// TIA Portal V16 export
// export: Created 2022-09-01T13:58:51.8751528Z, ExportSetting WithDefaults, DisplayName Totally Integrated Automation Portal, DisplayVersion V16, DisplayName TIA Portal Version Control Interface, DisplayVersion V16, DisplayName TIA Portal Openness, DisplayVersion V16, DisplayName STEP 7 Professional, DisplayVersion V16, DisplayName STEP 7 Safety, DisplayVersion V16, DisplayName WinCC Advanced, DisplayVersion V16
FUNCTION "Saídas_EV_Filt2" : Void   // FC5, LAD
{ S7_Optimized_Access := 'TRUE' }
VERSION : 0.1
// stored: AutoNumber true, IsIECCheckEnabled false, SetENOAutomatically false, UDAEnableTagReadback false
BEGIN

REGION Network 1
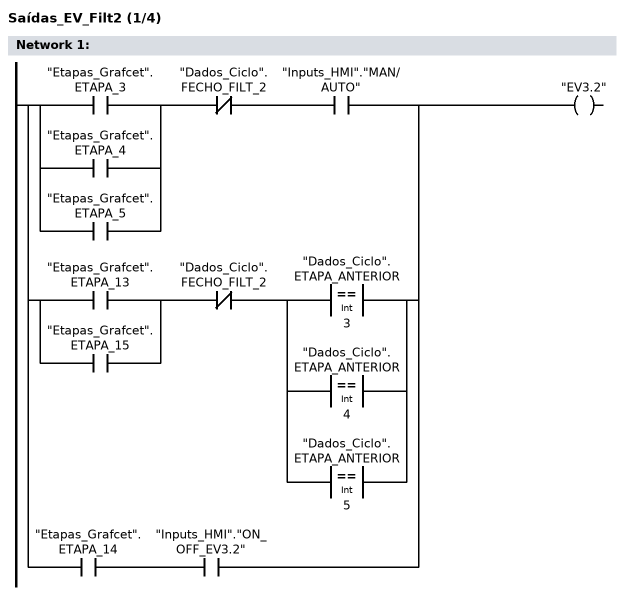
   RUNG wire#powerrail
      Contact( "Etapas_Grafcet".ETAPA_3 )
      wire#w1
      I_Contact( "Dados_Ciclo".FECHO_FILT_2 )
      Contact( "Inputs_HMI"."MAN/AUTO" )
      wire#w2
      Coil( "EV3.2" )
   END_RUNG
   RUNG wire#powerrail
      Contact( "Etapas_Grafcet".ETAPA_4 )
   END_RUNG wire#w1
   RUNG wire#powerrail
      Contact( "Etapas_Grafcet".ETAPA_5 )
   END_RUNG wire#w1
   RUNG wire#powerrail
      Contact( "Etapas_Grafcet".ETAPA_13 )
      wire#w3
      I_Contact( "Dados_Ciclo".FECHO_FILT_2 )
      wire#w4
      { S7_Templates := "SrcType := Int" } EQ_Contact(in1 := "Dados_Ciclo".ETAPA_ANTERIOR, in2 := 3)
   END_RUNG wire#w2
   RUNG wire#powerrail
      Contact( "Etapas_Grafcet".ETAPA_15 )
   END_RUNG wire#w3
   RUNG wire#w4
      { S7_Templates := "SrcType := Int" } EQ_Contact(in1 := "Dados_Ciclo".ETAPA_ANTERIOR, in2 := 4)
   END_RUNG wire#w2
   RUNG wire#w4
      { S7_Templates := "SrcType := Int" } EQ_Contact(in1 := "Dados_Ciclo".ETAPA_ANTERIOR, in2 := 5)
   END_RUNG wire#w2
   RUNG wire#powerrail
      Contact( "Etapas_Grafcet".ETAPA_14 )
      Contact( "Inputs_HMI"."ON_OFF_EV3.2" )
   END_RUNG wire#w2
   // the same network as SCL:
   "EV3.2" := (("Etapas_Grafcet".ETAPA_3 OR "Etapas_Grafcet".ETAPA_4 OR "Etapas_Grafcet".ETAPA_5) AND NOT "Dados_Ciclo".FECHO_FILT_2 AND "Inputs_HMI"."MAN/AUTO") OR (("Etapas_Grafcet".ETAPA_13 OR "Etapas_Grafcet".ETAPA_15) AND NOT "Dados_Ciclo".FECHO_FILT_2 AND (("Dados_Ciclo".ETAPA_ANTERIOR = 3) OR ("Dados_Ciclo".ETAPA_ANTERIOR = 4) OR ("Dados_Ciclo".ETAPA_ANTERIOR = 5))) OR ("Etapas_Grafcet".ETAPA_14 AND "Inputs_HMI"."ON_OFF_EV3.2");
END_REGION

REGION Network 2
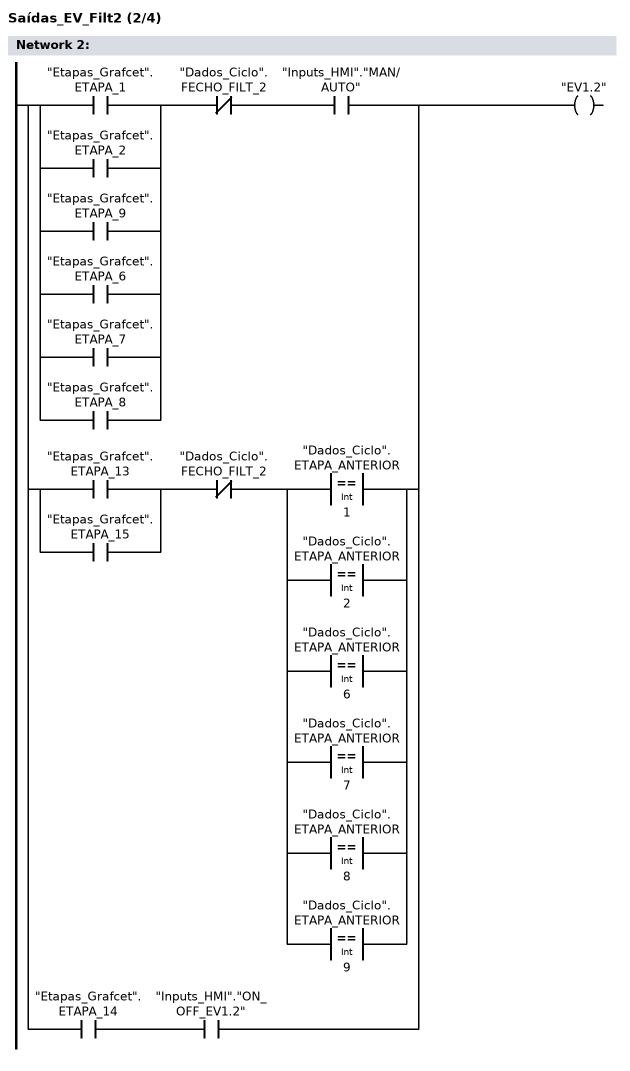
   RUNG wire#powerrail
      Contact( "Etapas_Grafcet".ETAPA_1 )
      wire#w1
      I_Contact( "Dados_Ciclo".FECHO_FILT_2 )
      Contact( "Inputs_HMI"."MAN/AUTO" )
      wire#w2
      Coil( "EV1.2" )
   END_RUNG
   RUNG wire#powerrail
      Contact( "Etapas_Grafcet".ETAPA_2 )
   END_RUNG wire#w1
   RUNG wire#powerrail
      Contact( "Etapas_Grafcet".ETAPA_9 )
   END_RUNG wire#w1
   RUNG wire#powerrail
      Contact( "Etapas_Grafcet".ETAPA_6 )
   END_RUNG wire#w1
   RUNG wire#powerrail
      Contact( "Etapas_Grafcet".ETAPA_7 )
   END_RUNG wire#w1
   RUNG wire#powerrail
      Contact( "Etapas_Grafcet".ETAPA_8 )
   END_RUNG wire#w1
   RUNG wire#powerrail
      Contact( "Etapas_Grafcet".ETAPA_13 )
      wire#w3
      I_Contact( "Dados_Ciclo".FECHO_FILT_2 )
      wire#w4
      { S7_Templates := "SrcType := Int" } EQ_Contact(in1 := "Dados_Ciclo".ETAPA_ANTERIOR, in2 := 1)
   END_RUNG wire#w2
   RUNG wire#powerrail
      Contact( "Etapas_Grafcet".ETAPA_15 )
   END_RUNG wire#w3
   RUNG wire#w4
      { S7_Templates := "SrcType := Int" } EQ_Contact(in1 := "Dados_Ciclo".ETAPA_ANTERIOR, in2 := 2)
   END_RUNG wire#w2
   RUNG wire#w4
      { S7_Templates := "SrcType := Int" } EQ_Contact(in1 := "Dados_Ciclo".ETAPA_ANTERIOR, in2 := 6)
   END_RUNG wire#w2
   RUNG wire#w4
      { S7_Templates := "SrcType := Int" } EQ_Contact(in1 := "Dados_Ciclo".ETAPA_ANTERIOR, in2 := 7)
   END_RUNG wire#w2
   RUNG wire#w4
      { S7_Templates := "SrcType := Int" } EQ_Contact(in1 := "Dados_Ciclo".ETAPA_ANTERIOR, in2 := 8)
   END_RUNG wire#w2
   RUNG wire#w4
      { S7_Templates := "SrcType := Int" } EQ_Contact(in1 := "Dados_Ciclo".ETAPA_ANTERIOR, in2 := 9)
   END_RUNG wire#w2
   RUNG wire#powerrail
      Contact( "Etapas_Grafcet".ETAPA_14 )
      Contact( "Inputs_HMI"."ON_OFF_EV1.2" )
   END_RUNG wire#w2
   // the same network as SCL:
   "EV1.2" := (("Etapas_Grafcet".ETAPA_1 OR "Etapas_Grafcet".ETAPA_2 OR "Etapas_Grafcet".ETAPA_9 OR "Etapas_Grafcet".ETAPA_6 OR "Etapas_Grafcet".ETAPA_7 OR "Etapas_Grafcet".ETAPA_8) AND NOT "Dados_Ciclo".FECHO_FILT_2 AND "Inputs_HMI"."MAN/AUTO") OR (("Etapas_Grafcet".ETAPA_13 OR "Etapas_Grafcet".ETAPA_15) AND NOT "Dados_Ciclo".FECHO_FILT_2 AND (("Dados_Ciclo".ETAPA_ANTERIOR = 1) OR ("Dados_Ciclo".ETAPA_ANTERIOR = 2) OR ("Dados_Ciclo".ETAPA_ANTERIOR = 6) OR ("Dados_Ciclo".ETAPA_ANTERIOR = 7) OR ("Dados_Ciclo".ETAPA_ANTERIOR = 8) OR ("Dados_Ciclo".ETAPA_ANTERIOR = 9))) OR ("Etapas_Grafcet".ETAPA_14 AND "Inputs_HMI"."ON_OFF_EV1.2");
END_REGION

REGION Network 3
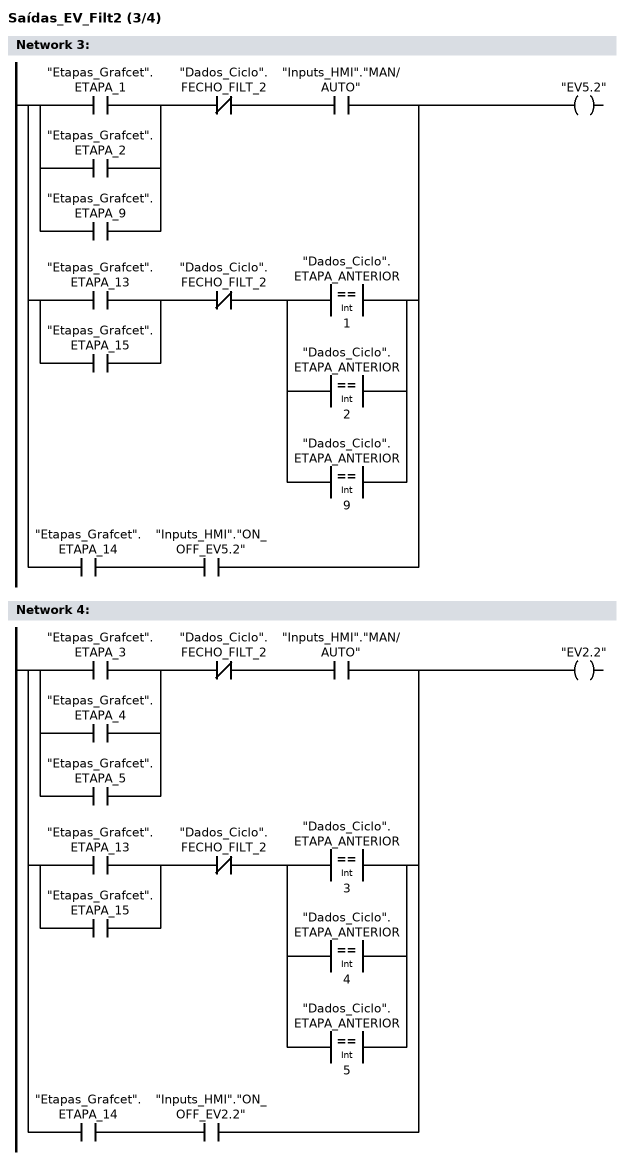
   RUNG wire#powerrail
      Contact( "Etapas_Grafcet".ETAPA_1 )
      wire#w1
      I_Contact( "Dados_Ciclo".FECHO_FILT_2 )
      Contact( "Inputs_HMI"."MAN/AUTO" )
      wire#w2
      Coil( "EV5.2" )
   END_RUNG
   RUNG wire#powerrail
      Contact( "Etapas_Grafcet".ETAPA_2 )
   END_RUNG wire#w1
   RUNG wire#powerrail
      Contact( "Etapas_Grafcet".ETAPA_9 )
   END_RUNG wire#w1
   RUNG wire#powerrail
      Contact( "Etapas_Grafcet".ETAPA_13 )
      wire#w3
      I_Contact( "Dados_Ciclo".FECHO_FILT_2 )
      wire#w4
      { S7_Templates := "SrcType := Int" } EQ_Contact(in1 := "Dados_Ciclo".ETAPA_ANTERIOR, in2 := 1)
   END_RUNG wire#w2
   RUNG wire#powerrail
      Contact( "Etapas_Grafcet".ETAPA_15 )
   END_RUNG wire#w3
   RUNG wire#w4
      { S7_Templates := "SrcType := Int" } EQ_Contact(in1 := "Dados_Ciclo".ETAPA_ANTERIOR, in2 := 2)
   END_RUNG wire#w2
   RUNG wire#w4
      { S7_Templates := "SrcType := Int" } EQ_Contact(in1 := "Dados_Ciclo".ETAPA_ANTERIOR, in2 := 9)
   END_RUNG wire#w2
   RUNG wire#powerrail
      Contact( "Etapas_Grafcet".ETAPA_14 )
      Contact( "Inputs_HMI"."ON_OFF_EV5.2" )
   END_RUNG wire#w2
   // the same network as SCL:
   "EV5.2" := (("Etapas_Grafcet".ETAPA_1 OR "Etapas_Grafcet".ETAPA_2 OR "Etapas_Grafcet".ETAPA_9) AND NOT "Dados_Ciclo".FECHO_FILT_2 AND "Inputs_HMI"."MAN/AUTO") OR (("Etapas_Grafcet".ETAPA_13 OR "Etapas_Grafcet".ETAPA_15) AND NOT "Dados_Ciclo".FECHO_FILT_2 AND (("Dados_Ciclo".ETAPA_ANTERIOR = 1) OR ("Dados_Ciclo".ETAPA_ANTERIOR = 2) OR ("Dados_Ciclo".ETAPA_ANTERIOR = 9))) OR ("Etapas_Grafcet".ETAPA_14 AND "Inputs_HMI"."ON_OFF_EV5.2");
END_REGION

REGION Network 4
   RUNG wire#powerrail
      Contact( "Etapas_Grafcet".ETAPA_3 )
      wire#w1
      I_Contact( "Dados_Ciclo".FECHO_FILT_2 )
      Contact( "Inputs_HMI"."MAN/AUTO" )
      wire#w2
      Coil( "EV2.2" )
   END_RUNG
   RUNG wire#powerrail
      Contact( "Etapas_Grafcet".ETAPA_4 )
   END_RUNG wire#w1
   RUNG wire#powerrail
      Contact( "Etapas_Grafcet".ETAPA_5 )
   END_RUNG wire#w1
   RUNG wire#powerrail
      Contact( "Etapas_Grafcet".ETAPA_13 )
      wire#w3
      I_Contact( "Dados_Ciclo".FECHO_FILT_2 )
      wire#w4
      { S7_Templates := "SrcType := Int" } EQ_Contact(in1 := "Dados_Ciclo".ETAPA_ANTERIOR, in2 := 3)
   END_RUNG wire#w2
   RUNG wire#powerrail
      Contact( "Etapas_Grafcet".ETAPA_15 )
   END_RUNG wire#w3
   RUNG wire#w4
      { S7_Templates := "SrcType := Int" } EQ_Contact(in1 := "Dados_Ciclo".ETAPA_ANTERIOR, in2 := 4)
   END_RUNG wire#w2
   RUNG wire#w4
      { S7_Templates := "SrcType := Int" } EQ_Contact(in1 := "Dados_Ciclo".ETAPA_ANTERIOR, in2 := 5)
   END_RUNG wire#w2
   RUNG wire#powerrail
      Contact( "Etapas_Grafcet".ETAPA_14 )
      Contact( "Inputs_HMI"."ON_OFF_EV2.2" )
   END_RUNG wire#w2
   // the same network as SCL:
   "EV2.2" := (("Etapas_Grafcet".ETAPA_3 OR "Etapas_Grafcet".ETAPA_4 OR "Etapas_Grafcet".ETAPA_5) AND NOT "Dados_Ciclo".FECHO_FILT_2 AND "Inputs_HMI"."MAN/AUTO") OR (("Etapas_Grafcet".ETAPA_13 OR "Etapas_Grafcet".ETAPA_15) AND NOT "Dados_Ciclo".FECHO_FILT_2 AND (("Dados_Ciclo".ETAPA_ANTERIOR = 3) OR ("Dados_Ciclo".ETAPA_ANTERIOR = 4) OR ("Dados_Ciclo".ETAPA_ANTERIOR = 5))) OR ("Etapas_Grafcet".ETAPA_14 AND "Inputs_HMI"."ON_OFF_EV2.2");
END_REGION

REGION Network 5
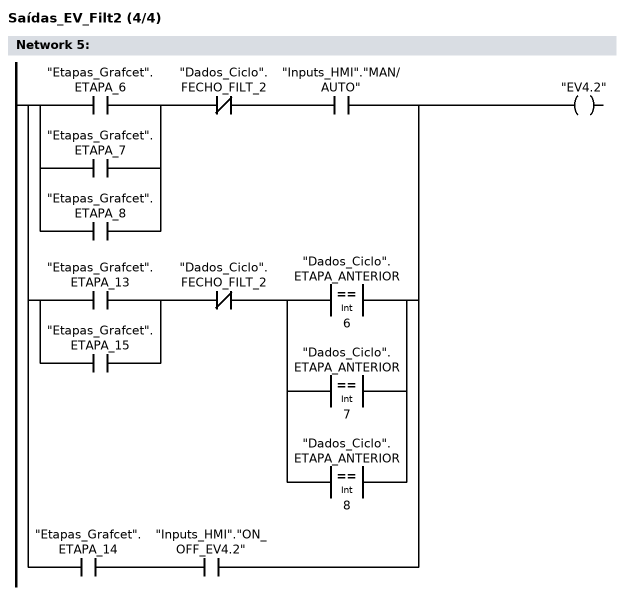
   RUNG wire#powerrail
      Contact( "Etapas_Grafcet".ETAPA_6 )
      wire#w1
      I_Contact( "Dados_Ciclo".FECHO_FILT_2 )
      Contact( "Inputs_HMI"."MAN/AUTO" )
      wire#w2
      Coil( "EV4.2" )
   END_RUNG
   RUNG wire#powerrail
      Contact( "Etapas_Grafcet".ETAPA_7 )
   END_RUNG wire#w1
   RUNG wire#powerrail
      Contact( "Etapas_Grafcet".ETAPA_8 )
   END_RUNG wire#w1
   RUNG wire#powerrail
      Contact( "Etapas_Grafcet".ETAPA_13 )
      wire#w3
      I_Contact( "Dados_Ciclo".FECHO_FILT_2 )
      wire#w4
      { S7_Templates := "SrcType := Int" } EQ_Contact(in1 := "Dados_Ciclo".ETAPA_ANTERIOR, in2 := 6)
   END_RUNG wire#w2
   RUNG wire#powerrail
      Contact( "Etapas_Grafcet".ETAPA_15 )
   END_RUNG wire#w3
   RUNG wire#w4
      { S7_Templates := "SrcType := Int" } EQ_Contact(in1 := "Dados_Ciclo".ETAPA_ANTERIOR, in2 := 7)
   END_RUNG wire#w2
   RUNG wire#w4
      { S7_Templates := "SrcType := Int" } EQ_Contact(in1 := "Dados_Ciclo".ETAPA_ANTERIOR, in2 := 8)
   END_RUNG wire#w2
   RUNG wire#powerrail
      Contact( "Etapas_Grafcet".ETAPA_14 )
      Contact( "Inputs_HMI"."ON_OFF_EV4.2" )
   END_RUNG wire#w2
   // the same network as SCL:
   "EV4.2" := (("Etapas_Grafcet".ETAPA_6 OR "Etapas_Grafcet".ETAPA_7 OR "Etapas_Grafcet".ETAPA_8) AND NOT "Dados_Ciclo".FECHO_FILT_2 AND "Inputs_HMI"."MAN/AUTO") OR (("Etapas_Grafcet".ETAPA_13 OR "Etapas_Grafcet".ETAPA_15) AND NOT "Dados_Ciclo".FECHO_FILT_2 AND (("Dados_Ciclo".ETAPA_ANTERIOR = 6) OR ("Dados_Ciclo".ETAPA_ANTERIOR = 7) OR ("Dados_Ciclo".ETAPA_ANTERIOR = 8))) OR ("Etapas_Grafcet".ETAPA_14 AND "Inputs_HMI"."ON_OFF_EV4.2");
END_REGION
END_FUNCTION
